INTERFACE IBaseSignal EXTENDS IOut

METHOD Control : IOut
VAR_INPUT
    setpoint : LREAL;
END_VAR
END_METHOD

METHOD Update : ISignal
VAR_INPUT
    value : LREAL;
END_VAR
END_METHOD

END_INTERFACE

(* stored: Version 1.1.0.1
   Itf IBaseSignal: Id {aeeffa15-e2d7-4163-9256-f2dfded0522d}
   Method Control: Id {025969cc-e5f9-4512-b433-fecde6f7bba7}
   Method Update: Id {f0eb471c-499e-499d-ae67-4a3bd890b28a} *)
